// TIA Portal V18 export
// export: Created 2026-04-18T00:00:00Z, ExportSetting WithDefaults
FUNCTION "FC_SCADA_Simulation" : Void   // FC10, LAD
{ S7_Optimized_Access := 'TRUE' }
VERSION : 0.1
// stored: AutoNumber true, IsIECCheckEnabled false
BEGIN

REGION Network 1: Tạo xung kích hoạt chu kỳ mô phỏng (50ms)
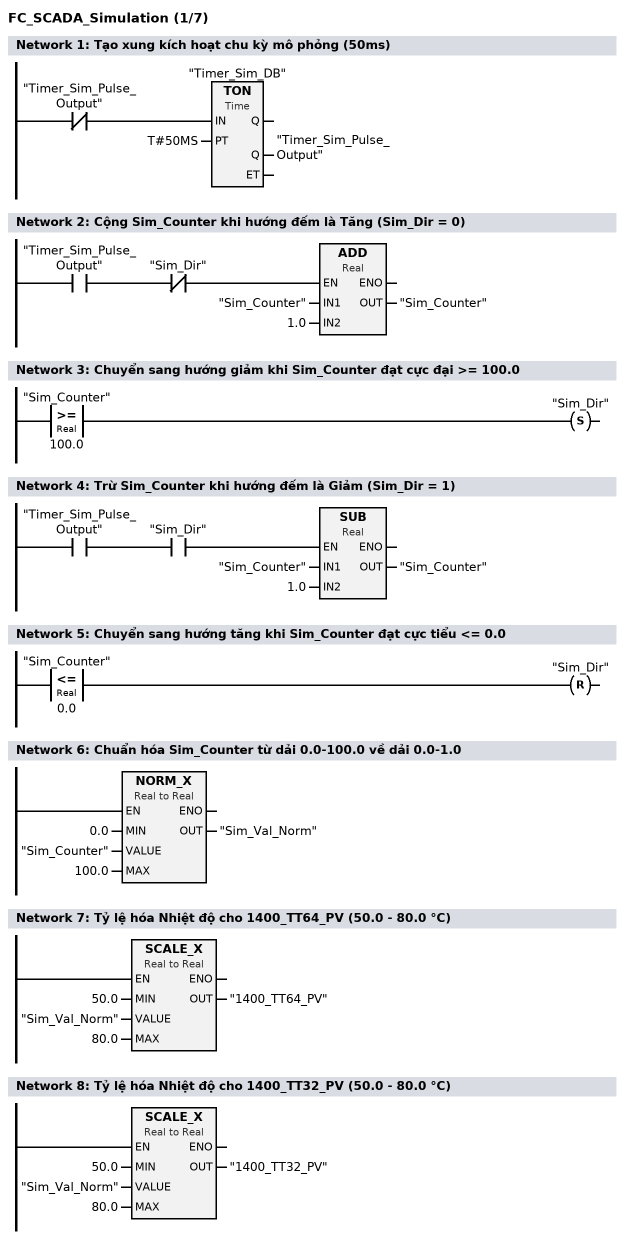
   RUNG wire#powerrail
      I_Contact( "Timer_Sim_Pulse_Output" )
      { S7_Templates := "time_type := Time" } "Timer_Sim_DB".TON(pt := T#50MS, q => "Timer_Sim_Pulse_Output", et =>)
   END_RUNG
   // the same network as SCL:
   "Timer_Sim_DB".TON(IN := NOT "Timer_Sim_Pulse_Output", PT := T#50MS, Q => "Timer_Sim_Pulse_Output");
END_REGION

REGION Network 2: Cộng Sim_Counter khi hướng đếm là Tăng (Sim_Dir = 0)
   RUNG wire#powerrail
      Contact( "Timer_Sim_Pulse_Output" )
      I_Contact( "Sim_Dir" )
      { S7_Templates := "SrcType := Real"; S7_GenerateENO := "TRUE" } Add(in1 := "Sim_Counter", in2 := 1.0, out => "Sim_Counter")
   END_RUNG
   // the same network as SCL:
   IF "Timer_Sim_Pulse_Output" AND NOT "Sim_Dir" THEN "Sim_Counter" := "Sim_Counter" + 1.0; END_IF;
END_REGION

REGION Network 3: Chuyển sang hướng giảm khi Sim_Counter đạt cực đại >= 100.0
   RUNG wire#powerrail
      { S7_Templates := "SrcType := Real" } GE_Contact(in1 := "Sim_Counter", in2 := 100.0)
      S_Coil( "Sim_Dir" )
   END_RUNG
   // the same network as SCL:
   IF "Sim_Counter" >= 100.0 THEN "Sim_Dir" := TRUE; END_IF;
END_REGION

REGION Network 4: Trừ Sim_Counter khi hướng đếm là Giảm (Sim_Dir = 1)
   RUNG wire#powerrail
      Contact( "Timer_Sim_Pulse_Output" )
      Contact( "Sim_Dir" )
      { S7_Templates := "SrcType := Real"; S7_GenerateENO := "TRUE" } Sub(in1 := "Sim_Counter", in2 := 1.0, out => "Sim_Counter")
   END_RUNG
   // the same network as SCL:
   IF "Timer_Sim_Pulse_Output" AND "Sim_Dir" THEN "Sim_Counter" := "Sim_Counter" - 1.0; END_IF;
END_REGION

REGION Network 5: Chuyển sang hướng tăng khi Sim_Counter đạt cực tiểu <= 0.0
   RUNG wire#powerrail
      { S7_Templates := "SrcType := Real" } LE_Contact(in1 := "Sim_Counter", in2 := 0.0)
      R_Coil( "Sim_Dir" )
   END_RUNG
   // the same network as SCL:
   IF "Sim_Counter" <= 0.0 THEN "Sim_Dir" := FALSE; END_IF;
END_REGION

REGION Network 6: Chuẩn hóa Sim_Counter từ dải 0.0-100.0 về dải 0.0-1.0
   RUNG wire#powerrail
      { S7_Templates := "[SrcType := Real, DestType := Real]" } Normalize(min := 0.0, value := "Sim_Counter", max := 100.0, out => "Sim_Val_Norm")
   END_RUNG
   // the same network as SCL:
   "Sim_Val_Norm" := NORM_X(MIN := 0.0, VALUE := "Sim_Counter", MAX := 100.0);
END_REGION

REGION Network 7: Tỷ lệ hóa Nhiệt độ cho 1400_TT64_PV (50.0 - 80.0 °C)
   RUNG wire#powerrail
      { S7_Templates := "[SrcType := Real, DestType := Real]" } Scale(min := 50.0, value := "Sim_Val_Norm", max := 80.0, out => "1400_TT64_PV")
   END_RUNG
   // the same network as SCL:
   "1400_TT64_PV" := SCALE_X(MIN := 50.0, VALUE := "Sim_Val_Norm", MAX := 80.0);
END_REGION

REGION Network 8: Tỷ lệ hóa Nhiệt độ cho 1400_TT32_PV (50.0 - 80.0 °C)
   RUNG wire#powerrail
      { S7_Templates := "[SrcType := Real, DestType := Real]" } Scale(min := 50.0, value := "Sim_Val_Norm", max := 80.0, out => "1400_TT32_PV")
   END_RUNG
   // the same network as SCL:
   "1400_TT32_PV" := SCALE_X(MIN := 50.0, VALUE := "Sim_Val_Norm", MAX := 80.0);
END_REGION

REGION Network 9: Tỷ lệ hóa Nhiệt độ cho 1400_TT101_PV (50.0 - 80.0 °C)
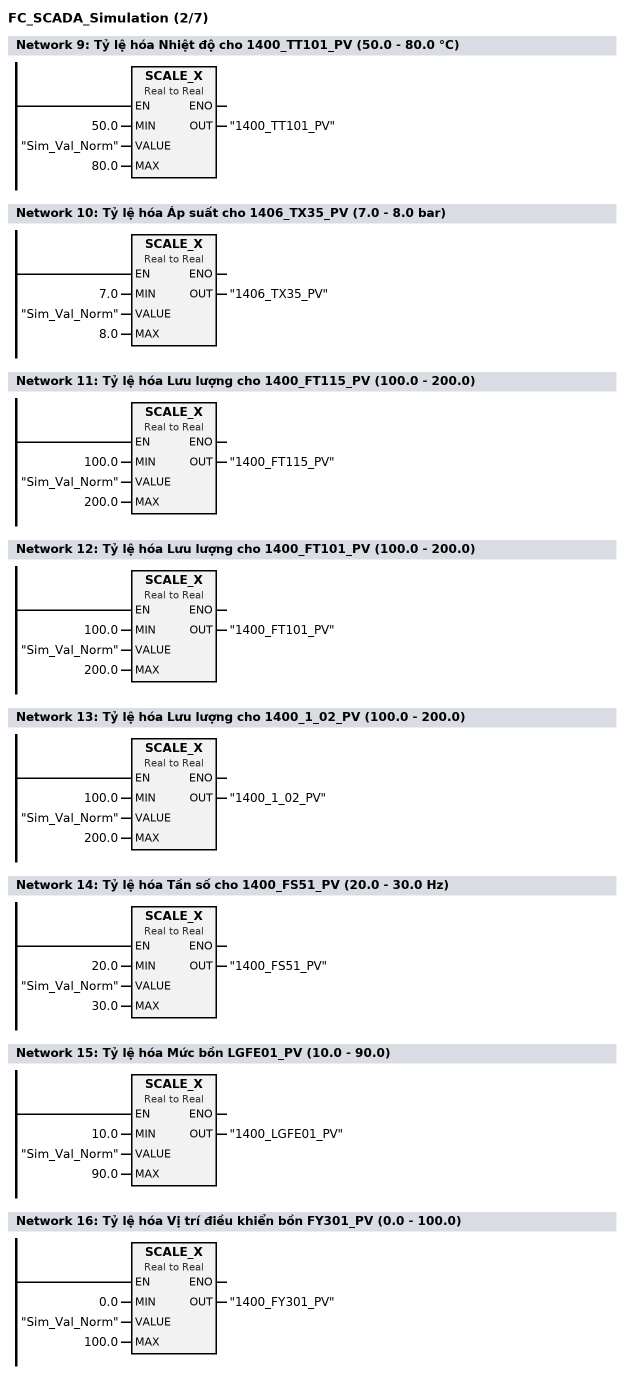
   RUNG wire#powerrail
      { S7_Templates := "[SrcType := Real, DestType := Real]" } Scale(min := 50.0, value := "Sim_Val_Norm", max := 80.0, out => "1400_TT101_PV")
   END_RUNG
   // the same network as SCL:
   "1400_TT101_PV" := SCALE_X(MIN := 50.0, VALUE := "Sim_Val_Norm", MAX := 80.0);
END_REGION

REGION Network 10: Tỷ lệ hóa Áp suất cho 1406_TX35_PV (7.0 - 8.0 bar)
   RUNG wire#powerrail
      { S7_Templates := "[SrcType := Real, DestType := Real]" } Scale(min := 7.0, value := "Sim_Val_Norm", max := 8.0, out => "1406_TX35_PV")
   END_RUNG
   // the same network as SCL:
   "1406_TX35_PV" := SCALE_X(MIN := 7.0, VALUE := "Sim_Val_Norm", MAX := 8.0);
END_REGION

REGION Network 11: Tỷ lệ hóa Lưu lượng cho 1400_FT115_PV (100.0 - 200.0)
   RUNG wire#powerrail
      { S7_Templates := "[SrcType := Real, DestType := Real]" } Scale(min := 100.0, value := "Sim_Val_Norm", max := 200.0, out => "1400_FT115_PV")
   END_RUNG
   // the same network as SCL:
   "1400_FT115_PV" := SCALE_X(MIN := 100.0, VALUE := "Sim_Val_Norm", MAX := 200.0);
END_REGION

REGION Network 12: Tỷ lệ hóa Lưu lượng cho 1400_FT101_PV (100.0 - 200.0)
   RUNG wire#powerrail
      { S7_Templates := "[SrcType := Real, DestType := Real]" } Scale(min := 100.0, value := "Sim_Val_Norm", max := 200.0, out => "1400_FT101_PV")
   END_RUNG
   // the same network as SCL:
   "1400_FT101_PV" := SCALE_X(MIN := 100.0, VALUE := "Sim_Val_Norm", MAX := 200.0);
END_REGION

REGION Network 13: Tỷ lệ hóa Lưu lượng cho 1400_1_02_PV (100.0 - 200.0)
   RUNG wire#powerrail
      { S7_Templates := "[SrcType := Real, DestType := Real]" } Scale(min := 100.0, value := "Sim_Val_Norm", max := 200.0, out => "1400_1_02_PV")
   END_RUNG
   // the same network as SCL:
   "1400_1_02_PV" := SCALE_X(MIN := 100.0, VALUE := "Sim_Val_Norm", MAX := 200.0);
END_REGION

REGION Network 14: Tỷ lệ hóa Tần số cho 1400_FS51_PV (20.0 - 30.0 Hz)
   RUNG wire#powerrail
      { S7_Templates := "[SrcType := Real, DestType := Real]" } Scale(min := 20.0, value := "Sim_Val_Norm", max := 30.0, out => "1400_FS51_PV")
   END_RUNG
   // the same network as SCL:
   "1400_FS51_PV" := SCALE_X(MIN := 20.0, VALUE := "Sim_Val_Norm", MAX := 30.0);
END_REGION

REGION Network 15: Tỷ lệ hóa Mức bồn LGFE01_PV (10.0 - 90.0)
   RUNG wire#powerrail
      { S7_Templates := "[SrcType := Real, DestType := Real]" } Scale(min := 10.0, value := "Sim_Val_Norm", max := 90.0, out => "1400_LGFE01_PV")
   END_RUNG
   // the same network as SCL:
   "1400_LGFE01_PV" := SCALE_X(MIN := 10.0, VALUE := "Sim_Val_Norm", MAX := 90.0);
END_REGION

REGION Network 16: Tỷ lệ hóa Vị trí điều khiển bồn FY301_PV (0.0 - 100.0)
   RUNG wire#powerrail
      { S7_Templates := "[SrcType := Real, DestType := Real]" } Scale(min := 0.0, value := "Sim_Val_Norm", max := 100.0, out => "1400_FY301_PV")
   END_RUNG
   // the same network as SCL:
   "1400_FY301_PV" := SCALE_X(MIN := 0.0, VALUE := "Sim_Val_Norm", MAX := 100.0);
END_REGION

REGION Network 17: Tỷ lệ hóa FTT02_PV (40.0 - 70.0)
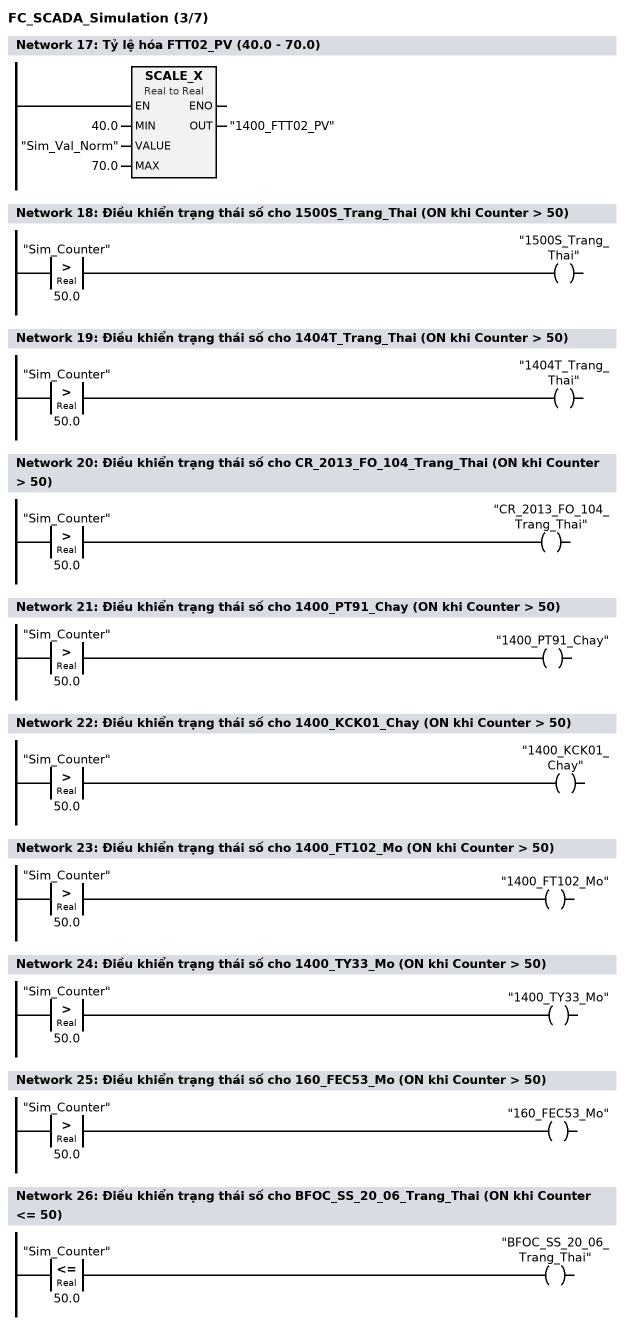
   RUNG wire#powerrail
      { S7_Templates := "[SrcType := Real, DestType := Real]" } Scale(min := 40.0, value := "Sim_Val_Norm", max := 70.0, out => "1400_FTT02_PV")
   END_RUNG
   // the same network as SCL:
   "1400_FTT02_PV" := SCALE_X(MIN := 40.0, VALUE := "Sim_Val_Norm", MAX := 70.0);
END_REGION

REGION Network 18: Điều khiển trạng thái số cho 1500S_Trang_Thai (ON khi Counter > 50)
   RUNG wire#powerrail
      { S7_Templates := "SrcType := Real" } GT_Contact(in1 := "Sim_Counter", in2 := 50.0)
      Coil( "1500S_Trang_Thai" )
   END_RUNG
   // the same network as SCL:
   "1500S_Trang_Thai" := "Sim_Counter" > 50.0;
END_REGION

REGION Network 19: Điều khiển trạng thái số cho 1404T_Trang_Thai (ON khi Counter > 50)
   RUNG wire#powerrail
      { S7_Templates := "SrcType := Real" } GT_Contact(in1 := "Sim_Counter", in2 := 50.0)
      Coil( "1404T_Trang_Thai" )
   END_RUNG
   // the same network as SCL:
   "1404T_Trang_Thai" := "Sim_Counter" > 50.0;
END_REGION

REGION Network 20: Điều khiển trạng thái số cho CR_2013_FO_104_Trang_Thai (ON khi Counter > 50)
   RUNG wire#powerrail
      { S7_Templates := "SrcType := Real" } GT_Contact(in1 := "Sim_Counter", in2 := 50.0)
      Coil( "CR_2013_FO_104_Trang_Thai" )
   END_RUNG
   // the same network as SCL:
   "CR_2013_FO_104_Trang_Thai" := "Sim_Counter" > 50.0;
END_REGION

REGION Network 21: Điều khiển trạng thái số cho 1400_PT91_Chay (ON khi Counter > 50)
   RUNG wire#powerrail
      { S7_Templates := "SrcType := Real" } GT_Contact(in1 := "Sim_Counter", in2 := 50.0)
      Coil( "1400_PT91_Chay" )
   END_RUNG
   // the same network as SCL:
   "1400_PT91_Chay" := "Sim_Counter" > 50.0;
END_REGION

REGION Network 22: Điều khiển trạng thái số cho 1400_KCK01_Chay (ON khi Counter > 50)
   RUNG wire#powerrail
      { S7_Templates := "SrcType := Real" } GT_Contact(in1 := "Sim_Counter", in2 := 50.0)
      Coil( "1400_KCK01_Chay" )
   END_RUNG
   // the same network as SCL:
   "1400_KCK01_Chay" := "Sim_Counter" > 50.0;
END_REGION

REGION Network 23: Điều khiển trạng thái số cho 1400_FT102_Mo (ON khi Counter > 50)
   RUNG wire#powerrail
      { S7_Templates := "SrcType := Real" } GT_Contact(in1 := "Sim_Counter", in2 := 50.0)
      Coil( "1400_FT102_Mo" )
   END_RUNG
   // the same network as SCL:
   "1400_FT102_Mo" := "Sim_Counter" > 50.0;
END_REGION

REGION Network 24: Điều khiển trạng thái số cho 1400_TY33_Mo (ON khi Counter > 50)
   RUNG wire#powerrail
      { S7_Templates := "SrcType := Real" } GT_Contact(in1 := "Sim_Counter", in2 := 50.0)
      Coil( "1400_TY33_Mo" )
   END_RUNG
   // the same network as SCL:
   "1400_TY33_Mo" := "Sim_Counter" > 50.0;
END_REGION

REGION Network 25: Điều khiển trạng thái số cho 160_FEC53_Mo (ON khi Counter > 50)
   RUNG wire#powerrail
      { S7_Templates := "SrcType := Real" } GT_Contact(in1 := "Sim_Counter", in2 := 50.0)
      Coil( "160_FEC53_Mo" )
   END_RUNG
   // the same network as SCL:
   "160_FEC53_Mo" := "Sim_Counter" > 50.0;
END_REGION

REGION Network 26: Điều khiển trạng thái số cho BFOC_SS_20_06_Trang_Thai (ON khi Counter <= 50)
   RUNG wire#powerrail
      { S7_Templates := "SrcType := Real" } LE_Contact(in1 := "Sim_Counter", in2 := 50.0)
      Coil( "BFOC_SS_20_06_Trang_Thai" )
   END_RUNG
   // the same network as SCL:
   "BFOC_SS_20_06_Trang_Thai" := "Sim_Counter" <= 50.0;
END_REGION

REGION Network 27: Điều khiển trạng thái số cho PC03010T01_Trang_Thai (ON khi Counter <= 50)
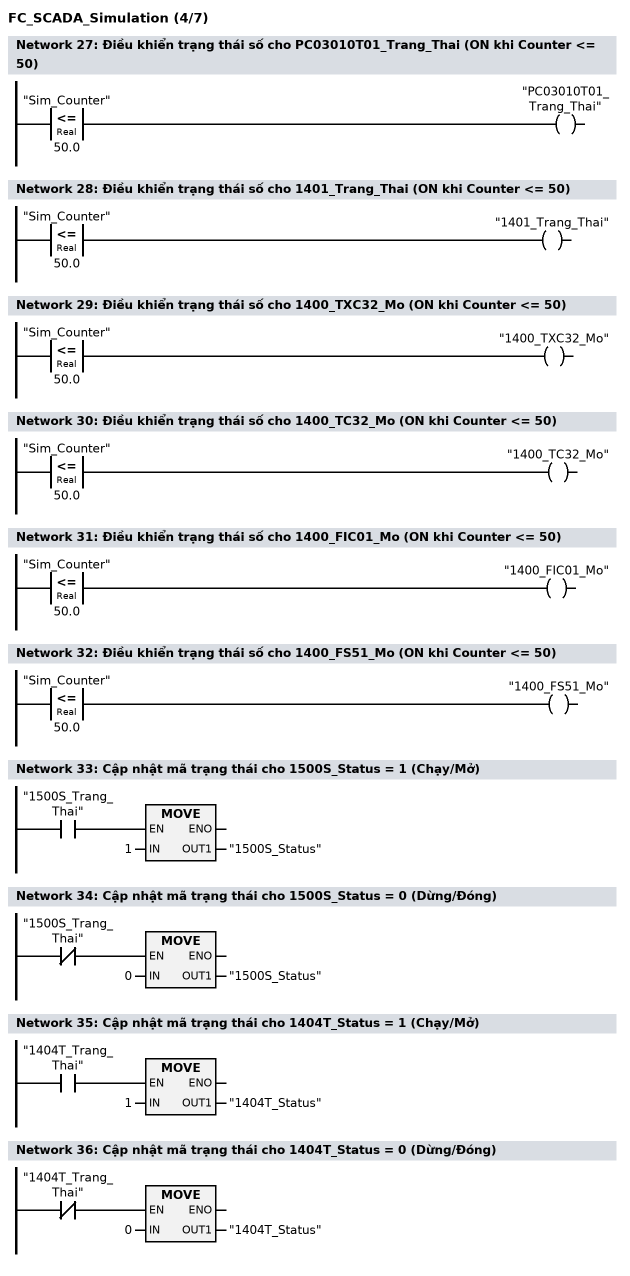
   RUNG wire#powerrail
      { S7_Templates := "SrcType := Real" } LE_Contact(in1 := "Sim_Counter", in2 := 50.0)
      Coil( "PC03010T01_Trang_Thai" )
   END_RUNG
   // the same network as SCL:
   "PC03010T01_Trang_Thai" := "Sim_Counter" <= 50.0;
END_REGION

REGION Network 28: Điều khiển trạng thái số cho 1401_Trang_Thai (ON khi Counter <= 50)
   RUNG wire#powerrail
      { S7_Templates := "SrcType := Real" } LE_Contact(in1 := "Sim_Counter", in2 := 50.0)
      Coil( "1401_Trang_Thai" )
   END_RUNG
   // the same network as SCL:
   "1401_Trang_Thai" := "Sim_Counter" <= 50.0;
END_REGION

REGION Network 29: Điều khiển trạng thái số cho 1400_TXC32_Mo (ON khi Counter <= 50)
   RUNG wire#powerrail
      { S7_Templates := "SrcType := Real" } LE_Contact(in1 := "Sim_Counter", in2 := 50.0)
      Coil( "1400_TXC32_Mo" )
   END_RUNG
   // the same network as SCL:
   "1400_TXC32_Mo" := "Sim_Counter" <= 50.0;
END_REGION

REGION Network 30: Điều khiển trạng thái số cho 1400_TC32_Mo (ON khi Counter <= 50)
   RUNG wire#powerrail
      { S7_Templates := "SrcType := Real" } LE_Contact(in1 := "Sim_Counter", in2 := 50.0)
      Coil( "1400_TC32_Mo" )
   END_RUNG
   // the same network as SCL:
   "1400_TC32_Mo" := "Sim_Counter" <= 50.0;
END_REGION

REGION Network 31: Điều khiển trạng thái số cho 1400_FIC01_Mo (ON khi Counter <= 50)
   RUNG wire#powerrail
      { S7_Templates := "SrcType := Real" } LE_Contact(in1 := "Sim_Counter", in2 := 50.0)
      Coil( "1400_FIC01_Mo" )
   END_RUNG
   // the same network as SCL:
   "1400_FIC01_Mo" := "Sim_Counter" <= 50.0;
END_REGION

REGION Network 32: Điều khiển trạng thái số cho 1400_FS51_Mo (ON khi Counter <= 50)
   RUNG wire#powerrail
      { S7_Templates := "SrcType := Real" } LE_Contact(in1 := "Sim_Counter", in2 := 50.0)
      Coil( "1400_FS51_Mo" )
   END_RUNG
   // the same network as SCL:
   "1400_FS51_Mo" := "Sim_Counter" <= 50.0;
END_REGION

REGION Network 33: Cập nhật mã trạng thái cho 1500S_Status = 1 (Chạy/Mở)
   RUNG wire#powerrail
      Contact( "1500S_Trang_Thai" )
      { S7_GenerateENO := "TRUE" } Move(in := 1, out1 => "1500S_Status")
   END_RUNG
   // the same network as SCL:
   IF "1500S_Trang_Thai" THEN "1500S_Status" := 1; END_IF;
END_REGION

REGION Network 34: Cập nhật mã trạng thái cho 1500S_Status = 0 (Dừng/Đóng)
   RUNG wire#powerrail
      I_Contact( "1500S_Trang_Thai" )
      { S7_GenerateENO := "TRUE" } Move(in := 0, out1 => "1500S_Status")
   END_RUNG
   // the same network as SCL:
   IF NOT "1500S_Trang_Thai" THEN "1500S_Status" := 0; END_IF;
END_REGION

REGION Network 35: Cập nhật mã trạng thái cho 1404T_Status = 1 (Chạy/Mở)
   RUNG wire#powerrail
      Contact( "1404T_Trang_Thai" )
      { S7_GenerateENO := "TRUE" } Move(in := 1, out1 => "1404T_Status")
   END_RUNG
   // the same network as SCL:
   IF "1404T_Trang_Thai" THEN "1404T_Status" := 1; END_IF;
END_REGION

REGION Network 36: Cập nhật mã trạng thái cho 1404T_Status = 0 (Dừng/Đóng)
   RUNG wire#powerrail
      I_Contact( "1404T_Trang_Thai" )
      { S7_GenerateENO := "TRUE" } Move(in := 0, out1 => "1404T_Status")
   END_RUNG
   // the same network as SCL:
   IF NOT "1404T_Trang_Thai" THEN "1404T_Status" := 0; END_IF;
END_REGION

REGION Network 37: Cập nhật mã trạng thái cho CR_2013_FO_104_Status = 1 (Chạy/Mở)
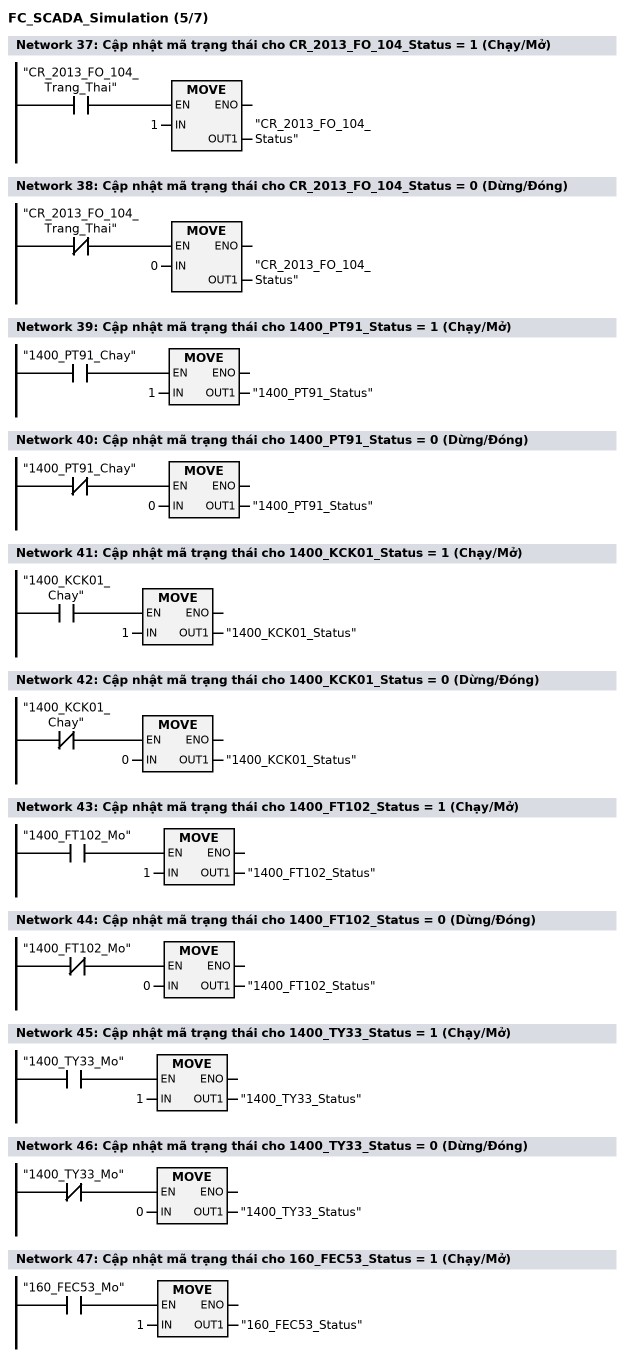
   RUNG wire#powerrail
      Contact( "CR_2013_FO_104_Trang_Thai" )
      { S7_GenerateENO := "TRUE" } Move(in := 1, out1 => "CR_2013_FO_104_Status")
   END_RUNG
   // the same network as SCL:
   IF "CR_2013_FO_104_Trang_Thai" THEN "CR_2013_FO_104_Status" := 1; END_IF;
END_REGION

REGION Network 38: Cập nhật mã trạng thái cho CR_2013_FO_104_Status = 0 (Dừng/Đóng)
   RUNG wire#powerrail
      I_Contact( "CR_2013_FO_104_Trang_Thai" )
      { S7_GenerateENO := "TRUE" } Move(in := 0, out1 => "CR_2013_FO_104_Status")
   END_RUNG
   // the same network as SCL:
   IF NOT "CR_2013_FO_104_Trang_Thai" THEN "CR_2013_FO_104_Status" := 0; END_IF;
END_REGION

REGION Network 39: Cập nhật mã trạng thái cho 1400_PT91_Status = 1 (Chạy/Mở)
   RUNG wire#powerrail
      Contact( "1400_PT91_Chay" )
      { S7_GenerateENO := "TRUE" } Move(in := 1, out1 => "1400_PT91_Status")
   END_RUNG
   // the same network as SCL:
   IF "1400_PT91_Chay" THEN "1400_PT91_Status" := 1; END_IF;
END_REGION

REGION Network 40: Cập nhật mã trạng thái cho 1400_PT91_Status = 0 (Dừng/Đóng)
   RUNG wire#powerrail
      I_Contact( "1400_PT91_Chay" )
      { S7_GenerateENO := "TRUE" } Move(in := 0, out1 => "1400_PT91_Status")
   END_RUNG
   // the same network as SCL:
   IF NOT "1400_PT91_Chay" THEN "1400_PT91_Status" := 0; END_IF;
END_REGION

REGION Network 41: Cập nhật mã trạng thái cho 1400_KCK01_Status = 1 (Chạy/Mở)
   RUNG wire#powerrail
      Contact( "1400_KCK01_Chay" )
      { S7_GenerateENO := "TRUE" } Move(in := 1, out1 => "1400_KCK01_Status")
   END_RUNG
   // the same network as SCL:
   IF "1400_KCK01_Chay" THEN "1400_KCK01_Status" := 1; END_IF;
END_REGION

REGION Network 42: Cập nhật mã trạng thái cho 1400_KCK01_Status = 0 (Dừng/Đóng)
   RUNG wire#powerrail
      I_Contact( "1400_KCK01_Chay" )
      { S7_GenerateENO := "TRUE" } Move(in := 0, out1 => "1400_KCK01_Status")
   END_RUNG
   // the same network as SCL:
   IF NOT "1400_KCK01_Chay" THEN "1400_KCK01_Status" := 0; END_IF;
END_REGION

REGION Network 43: Cập nhật mã trạng thái cho 1400_FT102_Status = 1 (Chạy/Mở)
   RUNG wire#powerrail
      Contact( "1400_FT102_Mo" )
      { S7_GenerateENO := "TRUE" } Move(in := 1, out1 => "1400_FT102_Status")
   END_RUNG
   // the same network as SCL:
   IF "1400_FT102_Mo" THEN "1400_FT102_Status" := 1; END_IF;
END_REGION

REGION Network 44: Cập nhật mã trạng thái cho 1400_FT102_Status = 0 (Dừng/Đóng)
   RUNG wire#powerrail
      I_Contact( "1400_FT102_Mo" )
      { S7_GenerateENO := "TRUE" } Move(in := 0, out1 => "1400_FT102_Status")
   END_RUNG
   // the same network as SCL:
   IF NOT "1400_FT102_Mo" THEN "1400_FT102_Status" := 0; END_IF;
END_REGION

REGION Network 45: Cập nhật mã trạng thái cho 1400_TY33_Status = 1 (Chạy/Mở)
   RUNG wire#powerrail
      Contact( "1400_TY33_Mo" )
      { S7_GenerateENO := "TRUE" } Move(in := 1, out1 => "1400_TY33_Status")
   END_RUNG
   // the same network as SCL:
   IF "1400_TY33_Mo" THEN "1400_TY33_Status" := 1; END_IF;
END_REGION

REGION Network 46: Cập nhật mã trạng thái cho 1400_TY33_Status = 0 (Dừng/Đóng)
   RUNG wire#powerrail
      I_Contact( "1400_TY33_Mo" )
      { S7_GenerateENO := "TRUE" } Move(in := 0, out1 => "1400_TY33_Status")
   END_RUNG
   // the same network as SCL:
   IF NOT "1400_TY33_Mo" THEN "1400_TY33_Status" := 0; END_IF;
END_REGION

REGION Network 47: Cập nhật mã trạng thái cho 160_FEC53_Status = 1 (Chạy/Mở)
   RUNG wire#powerrail
      Contact( "160_FEC53_Mo" )
      { S7_GenerateENO := "TRUE" } Move(in := 1, out1 => "160_FEC53_Status")
   END_RUNG
   // the same network as SCL:
   IF "160_FEC53_Mo" THEN "160_FEC53_Status" := 1; END_IF;
END_REGION

REGION Network 48: Cập nhật mã trạng thái cho 160_FEC53_Status = 0 (Dừng/Đóng)
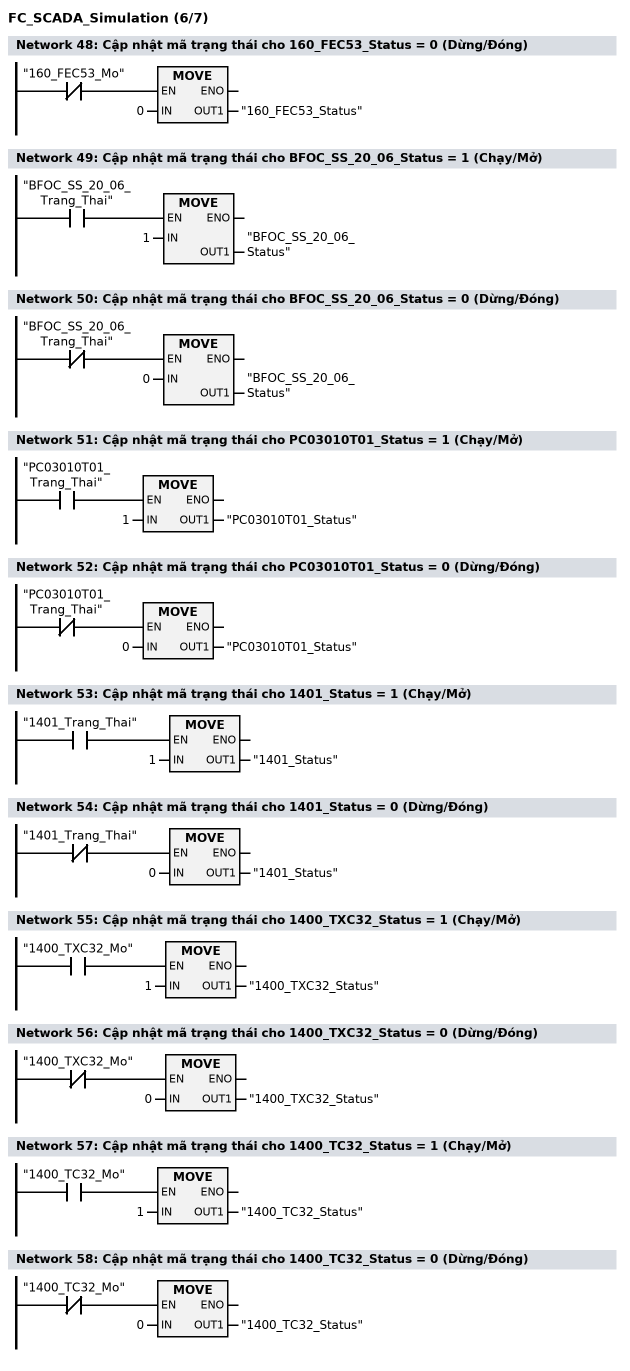
   RUNG wire#powerrail
      I_Contact( "160_FEC53_Mo" )
      { S7_GenerateENO := "TRUE" } Move(in := 0, out1 => "160_FEC53_Status")
   END_RUNG
   // the same network as SCL:
   IF NOT "160_FEC53_Mo" THEN "160_FEC53_Status" := 0; END_IF;
END_REGION

REGION Network 49: Cập nhật mã trạng thái cho BFOC_SS_20_06_Status = 1 (Chạy/Mở)
   RUNG wire#powerrail
      Contact( "BFOC_SS_20_06_Trang_Thai" )
      { S7_GenerateENO := "TRUE" } Move(in := 1, out1 => "BFOC_SS_20_06_Status")
   END_RUNG
   // the same network as SCL:
   IF "BFOC_SS_20_06_Trang_Thai" THEN "BFOC_SS_20_06_Status" := 1; END_IF;
END_REGION

REGION Network 50: Cập nhật mã trạng thái cho BFOC_SS_20_06_Status = 0 (Dừng/Đóng)
   RUNG wire#powerrail
      I_Contact( "BFOC_SS_20_06_Trang_Thai" )
      { S7_GenerateENO := "TRUE" } Move(in := 0, out1 => "BFOC_SS_20_06_Status")
   END_RUNG
   // the same network as SCL:
   IF NOT "BFOC_SS_20_06_Trang_Thai" THEN "BFOC_SS_20_06_Status" := 0; END_IF;
END_REGION

REGION Network 51: Cập nhật mã trạng thái cho PC03010T01_Status = 1 (Chạy/Mở)
   RUNG wire#powerrail
      Contact( "PC03010T01_Trang_Thai" )
      { S7_GenerateENO := "TRUE" } Move(in := 1, out1 => "PC03010T01_Status")
   END_RUNG
   // the same network as SCL:
   IF "PC03010T01_Trang_Thai" THEN "PC03010T01_Status" := 1; END_IF;
END_REGION

REGION Network 52: Cập nhật mã trạng thái cho PC03010T01_Status = 0 (Dừng/Đóng)
   RUNG wire#powerrail
      I_Contact( "PC03010T01_Trang_Thai" )
      { S7_GenerateENO := "TRUE" } Move(in := 0, out1 => "PC03010T01_Status")
   END_RUNG
   // the same network as SCL:
   IF NOT "PC03010T01_Trang_Thai" THEN "PC03010T01_Status" := 0; END_IF;
END_REGION

REGION Network 53: Cập nhật mã trạng thái cho 1401_Status = 1 (Chạy/Mở)
   RUNG wire#powerrail
      Contact( "1401_Trang_Thai" )
      { S7_GenerateENO := "TRUE" } Move(in := 1, out1 => "1401_Status")
   END_RUNG
   // the same network as SCL:
   IF "1401_Trang_Thai" THEN "1401_Status" := 1; END_IF;
END_REGION

REGION Network 54: Cập nhật mã trạng thái cho 1401_Status = 0 (Dừng/Đóng)
   RUNG wire#powerrail
      I_Contact( "1401_Trang_Thai" )
      { S7_GenerateENO := "TRUE" } Move(in := 0, out1 => "1401_Status")
   END_RUNG
   // the same network as SCL:
   IF NOT "1401_Trang_Thai" THEN "1401_Status" := 0; END_IF;
END_REGION

REGION Network 55: Cập nhật mã trạng thái cho 1400_TXC32_Status = 1 (Chạy/Mở)
   RUNG wire#powerrail
      Contact( "1400_TXC32_Mo" )
      { S7_GenerateENO := "TRUE" } Move(in := 1, out1 => "1400_TXC32_Status")
   END_RUNG
   // the same network as SCL:
   IF "1400_TXC32_Mo" THEN "1400_TXC32_Status" := 1; END_IF;
END_REGION

REGION Network 56: Cập nhật mã trạng thái cho 1400_TXC32_Status = 0 (Dừng/Đóng)
   RUNG wire#powerrail
      I_Contact( "1400_TXC32_Mo" )
      { S7_GenerateENO := "TRUE" } Move(in := 0, out1 => "1400_TXC32_Status")
   END_RUNG
   // the same network as SCL:
   IF NOT "1400_TXC32_Mo" THEN "1400_TXC32_Status" := 0; END_IF;
END_REGION

REGION Network 57: Cập nhật mã trạng thái cho 1400_TC32_Status = 1 (Chạy/Mở)
   RUNG wire#powerrail
      Contact( "1400_TC32_Mo" )
      { S7_GenerateENO := "TRUE" } Move(in := 1, out1 => "1400_TC32_Status")
   END_RUNG
   // the same network as SCL:
   IF "1400_TC32_Mo" THEN "1400_TC32_Status" := 1; END_IF;
END_REGION

REGION Network 58: Cập nhật mã trạng thái cho 1400_TC32_Status = 0 (Dừng/Đóng)
   RUNG wire#powerrail
      I_Contact( "1400_TC32_Mo" )
      { S7_GenerateENO := "TRUE" } Move(in := 0, out1 => "1400_TC32_Status")
   END_RUNG
   // the same network as SCL:
   IF NOT "1400_TC32_Mo" THEN "1400_TC32_Status" := 0; END_IF;
END_REGION

REGION Network 59: Cập nhật mã trạng thái cho 1400_FIC01_Status = 1 (Chạy/Mở)
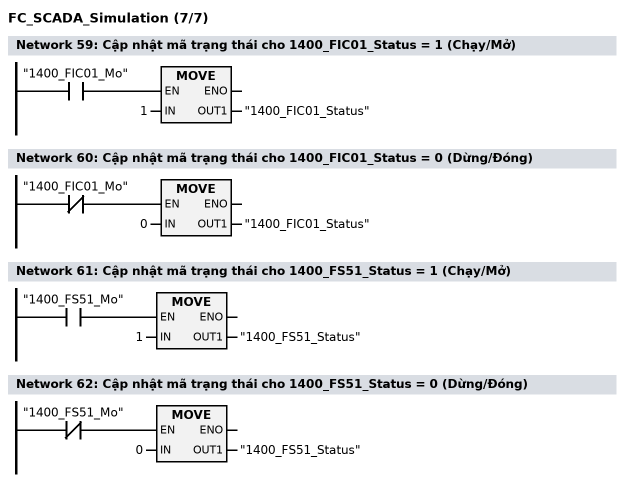
   RUNG wire#powerrail
      Contact( "1400_FIC01_Mo" )
      { S7_GenerateENO := "TRUE" } Move(in := 1, out1 => "1400_FIC01_Status")
   END_RUNG
   // the same network as SCL:
   IF "1400_FIC01_Mo" THEN "1400_FIC01_Status" := 1; END_IF;
END_REGION

REGION Network 60: Cập nhật mã trạng thái cho 1400_FIC01_Status = 0 (Dừng/Đóng)
   RUNG wire#powerrail
      I_Contact( "1400_FIC01_Mo" )
      { S7_GenerateENO := "TRUE" } Move(in := 0, out1 => "1400_FIC01_Status")
   END_RUNG
   // the same network as SCL:
   IF NOT "1400_FIC01_Mo" THEN "1400_FIC01_Status" := 0; END_IF;
END_REGION

REGION Network 61: Cập nhật mã trạng thái cho 1400_FS51_Status = 1 (Chạy/Mở)
   RUNG wire#powerrail
      Contact( "1400_FS51_Mo" )
      { S7_GenerateENO := "TRUE" } Move(in := 1, out1 => "1400_FS51_Status")
   END_RUNG
   // the same network as SCL:
   IF "1400_FS51_Mo" THEN "1400_FS51_Status" := 1; END_IF;
END_REGION

REGION Network 62: Cập nhật mã trạng thái cho 1400_FS51_Status = 0 (Dừng/Đóng)
   RUNG wire#powerrail
      I_Contact( "1400_FS51_Mo" )
      { S7_GenerateENO := "TRUE" } Move(in := 0, out1 => "1400_FS51_Status")
   END_RUNG
   // the same network as SCL:
   IF NOT "1400_FS51_Mo" THEN "1400_FS51_Status" := 0; END_IF;
END_REGION
END_FUNCTION
